Yaskawa INFORM job: R1_X(FRONIUS).JBI

/JOB
//NAME R1_X(FRONIUS)
///FOLDERNAME INNE
//POS
///NPOS 2,2,0,0,0,0
///TOOL 0
///POSTYPE PULSE
///PULSE
C00000=-133,28385,58033,-53,88656,-42
C00001=-240894,-52226,-3393,-234,41915,-81606
BC00000=67626,127399,695023
BC00001=381072,127399,695026
//INST
///DATE 2023/10/04 15:16
///ATTR SC,RW
///GROUP1 RB1,BS1
NOP
MOVJ C00000 BC00000 VJ=0.78
MOVJ C00001 BC00001 VJ=0.78
END
